PROGRAM prgMemPointerView
VAR
    pointerToMem:POINTER TO DWORD;  //DWORD
    offset: UDINT; //was UINT
	puls:R_TRIG; //only do stuff sometimes		

END_VAR
VAR // added by the converter: edge detectors and wires of the graphical bodies
    _rt1, _rt2, _rt3, _rt4 : R_TRIG;
END_VAR

//theme:VyJXkKWsxko

//buttons for adjusting offset, visu is keypad entry
actAdjustOffset();


//only do stuff every second
puls(clk:=System.OneSecond);

IF puls.Q THEN

	//move offset to keep global
	offset := ioView.memoffset * 4;
	
	//for M, MEMORY, MD, MW, Mx.y
	pointerToMem := ADR(%MD0);
	
	//add offset, from 0, add offset to desired memory location, e.g. "0 + 1024 = 1024" to view MD1024 and resulting areas
	pointerToMem := pointerToMem + offset;
	
	//limit value
	//pointerToMem := MIN(pointerToMem, 4294967295);
		
	//read values from raw pointer + offset
	MEMCPY(destAddr:=ADR(ioView.ViewingArray[0]), srcAddr:=pointerToMem + 0,n:=4);
	MEMCPY(destAddr:=ADR(ioView.ViewingArray[1]), srcAddr:=pointerToMem + 4,n:=4);
	MEMCPY(destAddr:=ADR(ioView.ViewingArray[2]), srcAddr:=pointerToMem + 8,n:=4);
	MEMCPY(destAddr:=ADR(ioView.ViewingArray[3]), srcAddr:=pointerToMem + 12,n:=4);
	MEMCPY(destAddr:=ADR(ioView.ViewingArray[4]), srcAddr:=pointerToMem + 16,n:=4);
	MEMCPY(destAddr:=ADR(ioView.ViewingArray[5]), srcAddr:=pointerToMem + 20,n:=4);
	MEMCPY(destAddr:=ADR(ioView.ViewingArray[6]), srcAddr:=pointerToMem + 24,n:=4);
	MEMCPY(destAddr:=ADR(ioView.ViewingArray[7]), srcAddr:=pointerToMem + 32,n:=4);
	MEMCPY(destAddr:=ADR(ioView.ViewingArray[8]), srcAddr:=pointerToMem + 36,n:=4);
	MEMCPY(destAddr:=ADR(ioView.ViewingArray[9]), srcAddr:=pointerToMem + 40,n:=4);
	MEMCPY(destAddr:=ADR(ioView.ViewingArray[10]), srcAddr:=pointerToMem + 44,n:=4);
	MEMCPY(destAddr:=ADR(ioView.ViewingArray[11]), srcAddr:=pointerToMem + 48,n:=4);
	MEMCPY(destAddr:=ADR(ioView.ViewingArray[12]), srcAddr:=pointerToMem + 52,n:=4);
	MEMCPY(destAddr:=ADR(ioView.ViewingArray[13]), srcAddr:=pointerToMem + 56,n:=4);
	MEMCPY(destAddr:=ADR(ioView.ViewingArray[14]), srcAddr:=pointerToMem + 60,n:=4);
	MEMCPY(destAddr:=ADR(ioView.ViewingArray[15]), srcAddr:=pointerToMem + 64,n:=4);
	
END_IF

ACTION actAdjustOffset:
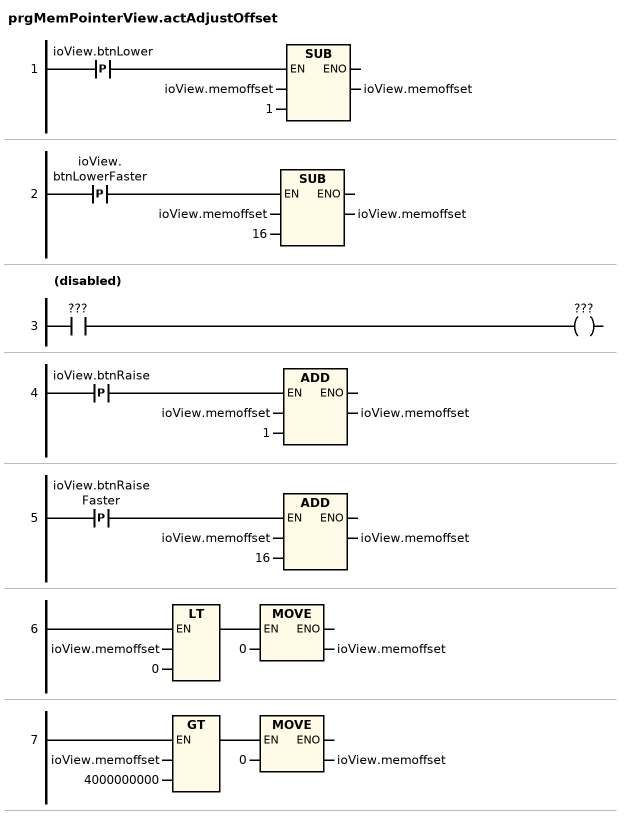
// NETWORK 1
_rt1(CLK := ioView.btnLower);
IF _rt1.Q THEN ioView.memoffset := ioView.memoffset - 1; END_IF

// NETWORK 2
_rt2(CLK := ioView.btnLowerFaster);
IF _rt2.Q THEN ioView.memoffset := ioView.memoffset - 16; END_IF

// NETWORK 3 (disabled)
// ??? := ???;

// NETWORK 4
_rt3(CLK := ioView.btnRaise);
IF _rt3.Q THEN ioView.memoffset := ioView.memoffset + 1; END_IF

// NETWORK 5
_rt4(CLK := ioView.btnRaiseFaster);
IF _rt4.Q THEN ioView.memoffset := ioView.memoffset + 16; END_IF

// NETWORK 6
IF ioView.memoffset < 0 THEN ioView.memoffset := 0; END_IF

// NETWORK 7
IF ioView.memoffset > 4000000000 THEN ioView.memoffset := 0; END_IF
END_ACTION

END_PROGRAM

(* stored: Version 1.1.0.1, ProductVersion 3.1.4024.12
   POU prgMemPointerView: Id {14ad67c0-13ff-42b6-871c-62e51a4859e1}, SpecialFunc None
   Action actAdjustOffset: Id {768519a0-735e-466b-9cc6-26b77674c384} *)
